// TIA Portal V19 export
VAR_GLOBAL   // PLC tag table "DIN"
END_VAR
